// TIA Portal V16 export
// export: Created 2022-09-01T14:29:18.0056747Z, ExportSetting WithDefaults, DisplayName Totally Integrated Automation Portal, DisplayVersion V16, DisplayName TIA Portal Version Control Interface, DisplayVersion V16, DisplayName TIA Portal Openness, DisplayVersion V16, DisplayName STEP 7 Professional, DisplayVersion V16, DisplayName STEP 7 Safety, DisplayVersion V16, DisplayName WinCC Advanced, DisplayVersion V16
FUNCTION "Níveis_TK02" : Void   // FC5, LAD
{ S7_Optimized_Access := 'TRUE' }
VERSION : 0.1
// stored: AutoNumber true, IsIECCheckEnabled false, SetENOAutomatically false, UDAEnableTagReadback false
BEGIN

REGION Network 1
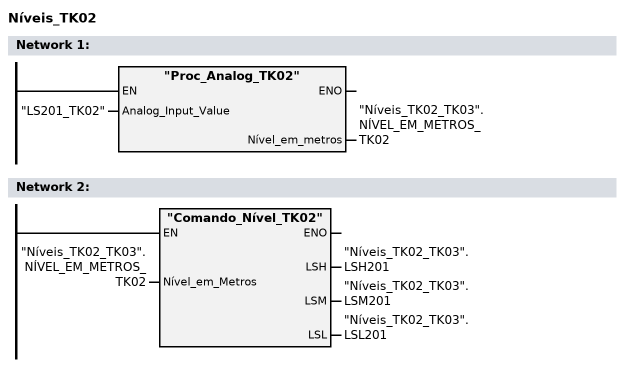
   RUNG wire#powerrail
      "Proc_Analog_TK02"(Analog_Input_Value := "LS201_TK02", Nível_em_metros => "Níveis_TK02_TK03".NÍVEL_EM_METROS_TK02)
   END_RUNG
   // the same network as SCL:
   "Proc_Analog_TK02"(Analog_Input_Value := "LS201_TK02",
                      Nível_em_metros => "Níveis_TK02_TK03".NÍVEL_EM_METROS_TK02);
END_REGION

REGION Network 2
   RUNG wire#powerrail
      "Comando_Nível_TK02"(Nível_em_Metros := "Níveis_TK02_TK03".NÍVEL_EM_METROS_TK02, LSH => "Níveis_TK02_TK03".LSH201, LSM => "Níveis_TK02_TK03".LSM201, LSL => "Níveis_TK02_TK03".LSL201)
   END_RUNG
   // the same network as SCL:
   "Comando_Nível_TK02"(Nível_em_Metros := "Níveis_TK02_TK03".NÍVEL_EM_METROS_TK02,
                        LSH => "Níveis_TK02_TK03".LSH201,
                        LSM => "Níveis_TK02_TK03".LSM201,
                        LSL => "Níveis_TK02_TK03".LSL201);
END_REGION
END_FUNCTION
